(* PLC project SafeLOGIC-2, BrAutomation SafeDESIGNER  4.2.6.2 *)
(* stored: companyURL http://www.br-automation.com, creationDateTime Mon Sep 25 14:20:17 2023 *)

PROGRAM Main

(* FBD diagram, written out as Structured Text *)
END_PROGRAM
